TYPE AllDataR :
	
// 	REGLES : 														
// 	Mettre seulement les structures des produits 					
// 	Séparer les Structures (Pas AX_PTR mais PTR_1, PTR_2, ...)		
// 	Les noms des variables sont globales (Pas ION7650 mais PM) 		 
//	PP
//	PTR_1, PTR_2, PTR_3
//	INV		

STRUCT
	
//PP               	
	PP					: PP;              	   (* PP *)
	
//SUB_MV               	
	SUBMV				: SUBMV_Exd;       	   (* SUB.MV*)

// PTR        	
	PTR					: ARRAY[1..CstNbPTR_G] OF  PTR_Exd;        (* PTR *)

//WS                	
	WS					: WS_AGMA;              		(* WS *)
                                           		
//COM                                      		
	SMS					: ServerSms;       		(* SMS      *)
	MAIL				: ServerMail;      		(* MAIL     *)
	COM					: COM_Status;	   		(* COM      *)
	CSV					: ServerCSV;       		(* CSV      *)
	CSVData				: LoggerCSV;       		(* CSVData  *) 
	
//OPC
	MesAlarmCode		: WORD ; 				 (* OPC Alarm Code   *)
	MesWarningCode		: WORD ; 				 (* OPC Warning Code *)
	MesEventCode : ARRAY[1..9] OF WORD ; //Akuo EventCode
END_STRUCT

END_TYPE

(* stored: Version 1.1.0.1, ProductVersion 3.1.4024.11
   DUT AllDataR: Id {af7c2bb0-329b-4ba0-9398-be02d4671aa9} *)
